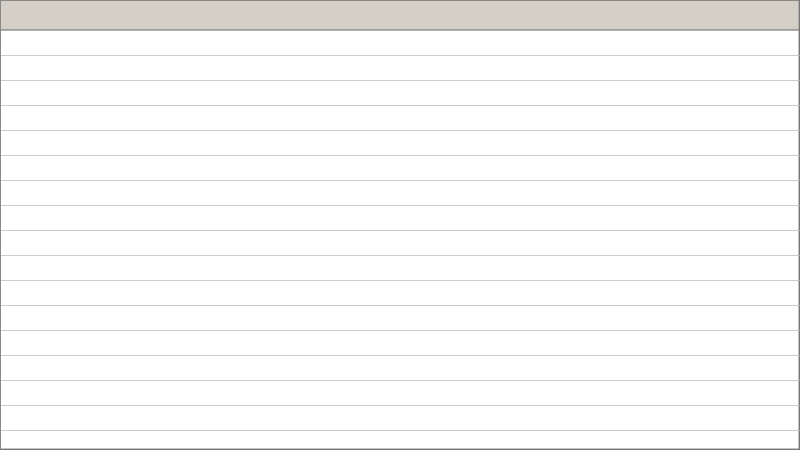
VISUALIZATION EventTableNew  // 800x450
VAR_IN_OUT
	arrEventData : ARRAY[1..512] OF ST_Event;
END_VAR
    Table (0,0 800x450)
END_VISUALIZATION

(* stored: Version 1.1.0.1, ProductVersion 3.1.4024.9
   Visu EventTableNew: Id {5c9a6bda-1880-4014-bd5b-48ce5849db5d} *)
